(* CODESYS project sensata_utilities.library
   Company: Sensata Technologies
   Version: 0.0.1
   DocFormat: reStructuredText
   Placeholder: Sensata_Utilities
   Title: Sensata_Utilities

Project tree, tasks and I/O mapping:
  libraries: Sensata_Common, * (Sensata Technologies); Tc2_Standard, * (Beckhoff Automation GmbH); Tc2_System, * (Beckhoff Automation GmbH); Tc2_Utilities, * (Beckhoff Automation GmbH); Tc3_JsonXml, * (Beckhoff Automation GmbH); Tc3_Module, * (Beckhoff Automation GmbH)
  Abstract/
    Obsolete/
      function block FB_DeviceAPI [ST]: M_Connect, M_Disconnect, M_GetConnectStatus, P_bConnectBusy, P_bConnected, M_CallMethod, M_GetProperty, P_bDeviceInterfaceBusy
    function block FB_CommandRouter [ST]: M_Connect, M_Disconnect, M_GetConnectStatus, P_bConnectBusy, P_bConnected, M_AwaitCommand, M_RequestRoute, M_RouteCommand, P_bCommandRoutingBusy
  Concrete/
    Obsolete/
      function block FB_AdsDeviceAPI [ST]: M_CallMethod, M_GetProperty, P_bDeviceInterfaceBusy
    function block FB_AdsCommandRouter [ST]: M_BuildMessage, M_ParseResult, M_RouteCommand, P_bCommandRoutingBusy
    function block FB_ApiParamBuilder [ST]: M_AddArrayElement, M_AddParameter, M_AddStructMember, M_ClearParameters, M_OutputToParameterList, M_Add, M_Pushback, M_ParseBool, M_ParseDateTime, M_ParseDouble, M_ParseInt, M_ParseInt64, M_ParseString, M_ParseUint, M_ParseUint64, M_GetArrayElement, M_GetParameter, M_GetStructMember, M_LoadFromParameterList
  DUTs/
    Obsolete/
      data type T_ApiMethodParameters
    data type E_AdsCommandRouterError
    data type ST_ApiParameter
    data type T_ApiMessage
    data type T_ApiParameterList
    data type T_ApiParamValue
  Globals/
    Obsolete/
      global variables GVL_DeviceAPI
    global variables GVL_Api
  Interfaces/
    Obsolete/
      interface I_DeviceInterface: M_CallMethod, M_GetProperty, P_bDeviceInterfaceBusy
      interface I_ModularAPI: M_CallMethod, P_bApiBusy
    interface I_CommandRouting: M_AwaitCommand, M_RequestRoute, M_RouteCommand, P_bCommandRoutingBusy
  Project Information/
    function F_GetCompany [ST]
    function F_GetTitle [ST]
    function F_GetVersion [ST]
  Version/
    global variables Global_Version
*)

// DUTs/Obsolete/T_ApiMethodParameters
{attribute 'obsolete' := 'Only used on obsolete FB_DeviceAPI'} 
TYPE T_ApiMethodParameters : 
	ARRAY [1..GVL_DeviceAPI.uintMAX_CALL_METHOD_PARAMETERS]
		OF ARRAY [1..2] OF Tc2_System.T_MaxString;
END_TYPE

// DUTs/E_AdsCommandRouterError
{attribute 'qualified_only'}
{attribute 'strict'}
TYPE E_AdsCommandRouterError :
(
	None := 0,
	IncorrectResponseFormat := 100,
	NoResponseReceived := 101,
	AdsError := 200,
	PointerError := 300
) UDINT;
END_TYPE

// DUTs/ST_ApiParameter
TYPE ST_ApiParameter :
STRUCT
	strKey : T_MaxString;
	strValue : T_ApiParamValue;
END_STRUCT
END_TYPE

// DUTs/T_ApiMessage
TYPE T_ApiMessage : STRING(GVL_Api.dintMSG_STRING_SIZE); END_TYPE

// DUTs/T_ApiParameterList
TYPE T_ApiParameterList : ARRAY[GVL_Api.dintPARAM_LOWER_BOUND..GVL_Api.dintPARAM_UPPER_BOUND] OF ST_ApiParameter; END_TYPE

// DUTs/T_ApiParamValue
TYPE T_ApiParamValue : STRING(GVL_Api.dintPARAM_STRING_SIZE); END_TYPE

// Globals/Obsolete/GVL_DeviceAPI
{attribute 'qualified_only'}
VAR_GLOBAL CONSTANT
	uintMAX_CALL_METHOD_PARAMETERS : UINT := 16;
END_VAR

// Globals/GVL_Api
{attribute 'qualified_only'}
VAR_GLOBAL CONSTANT
	dintPARAM_LOWER_BOUND : DINT := 0;
	dintPARAM_UPPER_BOUND : DINT := 31;
	dintPARAM_STRING_SIZE : DINT := 1023;
	dintMSG_STRING_SIZE : DINT := 4095;
END_VAR

// Version/Global_Version
{attribute 'TcGenerated'}
{attribute 'no-analysis'}
{attribute 'linkalways'}
// This function has been automatically generated from the project information.
VAR_GLOBAL CONSTANT
	{attribute 'const_non_replaced'}
	stLibVersion_Sensata_Utilities : ST_LibVersion := (iMajor := 0, iMinor := 0, iBuild := 1, iRevision := 0, nFlags := 0, sVersion := '0.0.1');
END_VAR

// Abstract/Obsolete/FB_DeviceAPI
(*
===============================================================================
Abstract Device API
===============================================================================
:Contact: Kevin Sanita <ksanita@sensata.com>
:Last Edited: March 2022

:Description: Represents a device API that allows for methods and
	properties to be called and accessed

:Notes:
* ``M_CallMethod`` to send a call method command to a device API
* ``M_GetProperty`` to send a get property command to a device API

:Change Log:
- **March 25, 2022** Initial version
*)
{attribute 'obsolete' := 'Use FB_CommandRouter instead!'} 
FUNCTION_BLOCK ABSTRACT FB_DeviceAPI EXTENDS FB_Module IMPLEMENTS I_DeviceInterface, I_Connectable
VAR_INPUT
END_VAR
VAR_OUTPUT
END_VAR
VAR
	bConnected: BOOL;
END_VAR

(* Connect to the device. *)
METHOD M_Connect : BOOL
bConnected := TRUE;
M_Connect := TRUE;
THIS^.M_LogWarning('M_Connect not implemented!');
END_METHOD

(* Disconnect from the camera. *)
METHOD M_Disconnect : BOOL
bConnected := FALSE;
M_Disconnect := TRUE;
THIS^.M_LogWarning('M_Disconnect not implemented!');
END_METHOD

(* Get the device connection status. *)
METHOD M_GetConnectStatus : BOOL
VAR_OUTPUT
	(* TRUE if the device is connected, FALSE otherwise. *)
	bConnected	: BOOL;
END_VAR
bConnected := THIS^.bConnected;
M_GetConnectStatus := TRUE;
END_METHOD

(* TRUE while the device is connecting or disconnecting. *)
PROPERTY P_bConnectBusy : BOOL
GET
P_bConnectBusy := FALSE;
END_GET
END_PROPERTY

(* TRUE if the camera is connected. *)
PROPERTY P_bConnected : BOOL
GET
P_bConnected := bConnected;
END_GET
END_PROPERTY

(* Calls a device method from a device API. *)
METHOD M_CallMethod : BOOL
VAR_INPUT
	(* UniqueID of the target module. *)
	strTargetId		: Tc2_System.T_MaxString;
	(* Name of the method to call. *)
	strMethodName	: Tc2_System.T_MaxString;
	(* 2D array of parameter name and parameter value. *)
	arrParameters	: T_ApiMethodParameters;
END_VAR
VAR_OUTPUT
	(* Return data of the method. *)
	strReturn	: Tc2_System.T_MaxString;
END_VAR
M_CallMethod := FALSE;
END_METHOD

(* Gets the value of a device property through an API. *)
METHOD M_GetProperty : BOOL
VAR_INPUT
	(* Name of the property to get. *)
	strPropertyName	: Tc2_System.T_MaxString;
END_VAR
VAR_OUTPUT
	(* Value of the property. *)
	strReturn	: Tc2_System.T_MaxString;
END_VAR
M_GetProperty := FALSE;
END_METHOD

(* True while a device interface command is running. *)
PROPERTY P_bDeviceInterfaceBusy : BOOL
GET
P_bDeviceInterfaceBusy := FALSE;
END_GET
END_PROPERTY

END_FUNCTION_BLOCK

// Abstract/FB_CommandRouter
FUNCTION_BLOCK FB_CommandRouter EXTENDS FB_Module
	IMPLEMENTS I_CommandRouting, I_Connectable
VAR_INPUT
END_VAR
VAR_OUTPUT
END_VAR
VAR
	cr_bConnected: BOOL;
END_VAR

(* This method should establish any external connections required to use the
	functions of the device, and return TRUE and set P_bConnected to TRUE once
	connected. *)
METHOD M_Connect : BOOL
THIS^.M_LogWarning('M_Connect not implemented!');
cr_bConnected := TRUE;
M_Connect := TRUE;
END_METHOD

(* This method should break any connections established by M_Connect. It should
	immediately set P_bConnected to false unless all connections are known to
	be still active, and return TRUE once those connections are all fully
	disconnected. *)
METHOD M_Disconnect : BOOL
THIS^.M_LogWarning('M_Disconnect not implemented!');
cr_bConnected := FALSE;
M_Disconnect := TRUE;
END_METHOD

(* This method should explicitly check the connection status of the device.
	Once the connection status is known, this method should return TRUE.
	If this method fails, P_bConnected should be set to FALSE since the device
	is not absolutely known to still be connected. *)
METHOD M_GetConnectStatus : BOOL
VAR_OUTPUT
	(* This should return TRUE if all connections required to make the device
		function properly are known to be connected, and FALSE otherwise. *)
	bConnected	: BOOL;
END_VAR
THIS^.M_LogWarning('M_GetConnectStatus not implemented!');
M_GetConnectStatus := TRUE;
bConnected := cr_bConnected;
END_METHOD

(* This property should be TRUE while any method in this interface is actively
	executing, or FALSE otherwise. *)
PROPERTY P_bConnectBusy : BOOL
GET
P_bConnectBusy := FALSE;
END_GET
END_PROPERTY

(* This should be set to TRUE if M_Connect is successful or M_GetConnectStatus
	determines the device to be connected, and set to FALSE if M_Disconnect is
	called at all, M_GetConnectStatus fails, or M_GetConnectStatus determines
	the device to be not connected. *)
PROPERTY P_bConnected : BOOL
GET
P_bConnected := cr_bConnected;
END_GET
END_PROPERTY

(* Waits for the command with the given route ID to complete. *)
METHOD M_AwaitCommand : BOOL
VAR_INPUT
	(* ID assigned to the route. *)
	_in_udintRouteId	: UDINT;
	(* Timeout time for the command. *)
	_in_timeTimeout	: TIME;
END_VAR
VAR_IN_OUT
	(* Array of data key:value pairs. This will be filled with output
		data on command success. This is required due to memory limitations
		within Beckhoff. *)
	_inout_arrOutputs	: T_ApiParameterList;
END_VAR
VAR_OUTPUT
	(* True if the command executed without error. Does not necessarily
	mean the command performed the task it was expected to perform, just
	means that the method returned a value. *)
	_out_bCommandExecuted	: BOOL;
	(* The return value of the method. *)
	_out_strReturnValue	: T_ApiParamValue;
END_VAR
THIS^.M_LogWarning('M_AwaitCommand not implemented!');
M_AwaitCommand := TRUE;
END_METHOD

(* Sends a route request and returns a route ID if successfully routed. 
Use M_AwaitCommand with the route ID as input in order to wait for and get
the results of the routed command. *)
METHOD M_RequestRoute : BOOL
VAR_INPUT
	(* Unique ID of the module to call the command on. *)
	_in_strModuleId	: Tc2_System.T_MaxString;
	(* Name of the method to call. *)
	_in_strMethodName	: Tc2_System.T_MaxString;
	(* Timeout time for the route. *)
	_in_timeTimeout	: TIME;
END_VAR
VAR_IN_OUT
	(* Array of data key:value pairs. This should be set to the parameters
		of the command. *)
	_inout_arrParameters	: T_ApiParameterList;
END_VAR
VAR_OUTPUT
	(* ID assigned to the route. *)
	_out_udintRouteId	: UDINT;
END_VAR
THIS^.M_LogWarning('M_RequestRoute not implemented!');
M_RequestRoute := TRUE;
END_METHOD

(* Routes the given command and waits for the command to finish before
returning the output data of the command. *)
METHOD M_RouteCommand : BOOL
VAR_INPUT
	(* Unique ID of the module to call the command on. *)
	_in_strModuleId	: Tc2_System.T_MaxString;
	(* Name of the method to call. *)
	_in_strMethodName	: Tc2_System.T_MaxString;
	(* Timeout time for the command. *)
	_in_timeTimeout	: TIME;
END_VAR
VAR_IN_OUT
	(* Array of input parameter key:value pairs. *)
	_inout_arrParameters	: T_ApiParameterList;
	(* Array of output key:value pairs. Will be cleared and then populated with output data. *)
	_inout_arrOutputs	: T_ApiParameterList;
END_VAR
VAR_OUTPUT
	(* True if the command executed without error. Does not necessarily
	mean the command performed the task it was expected to perform, just
	means that the method returned a value. *)
	_out_bCommandExecuted	: BOOL;
	(* The return value of the method as a string. *)
	_out_strReturnValue	: T_ApiParamValue;
END_VAR
THIS^.M_LogWarning('M_RouteCommand not implemented!');
M_RouteCommand := TRUE;
END_METHOD

(* TRUE while any method in this interface is running. *)
PROPERTY P_bCommandRoutingBusy : BOOL
GET
P_bCommandRoutingBusy := TRUE;
END_GET
END_PROPERTY

END_FUNCTION_BLOCK

// Interfaces/I_CommandRouting
INTERFACE I_CommandRouting

(* Waits for the command with the given route ID to complete. *)
METHOD M_AwaitCommand : BOOL
VAR_INPUT
	(* ID assigned to the route. *)
	_in_udintRouteId : UDINT;
	
	(* Timeout time for the command. *)
	_in_timeTimeout : TIME;
END_VAR
VAR_IN_OUT
	(* Array of data key:value pairs. This will be filled with output
		data on command success. This is required due to memory limitations
		within Beckhoff. *)
	_inout_arrOutputs : T_ApiParameterList;
END_VAR
VAR_OUTPUT
	(* True if the command executed without error. Does not necessarily
	mean the command performed the task it was expected to perform, just
	means that the method returned a value. *)
	_out_bCommandExecuted : BOOL;
	
	(* The return value of the method. *)
	_out_strReturnValue : T_ApiParamValue;
END_VAR
END_METHOD

(* Sends a route request and returns a route ID if successfully routed. 
Use M_AwaitCommand with the route ID as input in order to wait for and get
the results of the routed command. *)
METHOD M_RequestRoute : BOOL
VAR_INPUT
	(* Unique ID of the module to call the command on. *)
	_in_strModuleId : T_MaxString;
	
	(* Name of the method to call. *)
	_in_strMethodName : T_MaxString;
	
	(* Timeout time for the route. *)
	_in_timeTimeout : TIME;
END_VAR
VAR_IN_OUT
	(* Array of data key:value pairs. This should be set to the parameters
		of the command. *)
	_inout_arrParameters : T_ApiParameterList;
END_VAR
VAR_OUTPUT
	(* ID assigned to the route. *)
	_out_udintRouteId : UDINT;
END_VAR
END_METHOD

(* Routes the given command and waits for the command to finish before
returning the output data of the command. *)
METHOD M_RouteCommand : BOOL
VAR_INPUT
	(* Unique ID of the module to call the command on. *)
	_in_strModuleId	: Tc2_System.T_MaxString;
	
	(* Name of the method to call. *)
	_in_strMethodName	: Tc2_System.T_MaxString;
	
	(* Timeout time for the command. *)
	_in_timeTimeout	: TIME;
END_VAR
VAR_IN_OUT
	(* Array of input parameter key:value pairs. *)
	_inout_arrParameters	: T_ApiParameterList;
	
	(* Array of output key:value pairs. Will be cleared and then populated with output data. *)
	_inout_arrOutputs	: T_ApiParameterList;
END_VAR
VAR_OUTPUT
	(* True if the command executed without error. Does not necessarily
	mean the command performed the task it was expected to perform, just
	means that the method returned a value. *)
	_out_bCommandExecuted	: BOOL;
	
	(* The return value of the method as a string. *)
	_out_strReturnValue	: T_ApiParamValue;
END_VAR
END_METHOD

(* TRUE while any method in this interface is running. *)
PROPERTY P_bCommandRoutingBusy : BOOL
GET
END_GET
END_PROPERTY

END_INTERFACE

// Interfaces/Obsolete/I_DeviceInterface
INTERFACE I_DeviceInterface

(* Calls a device method from a device API. *)
METHOD M_CallMethod : BOOL
VAR_INPUT
	(* UniqueID of the target module. *)
	strTargetId		: Tc2_System.T_MaxString;
		
	(* Name of the method to call. *)
	strMethodName : T_MaxString;
	
	(* 2D array of parameter name and parameter value. *)
	arrParameters : T_ApiMethodParameters;
END_VAR
VAR_OUTPUT
	(* Return data of the method. *)
	strReturn : T_MaxString;
END_VAR
END_METHOD

(* Gets the value of a device property through an API. *)
METHOD M_GetProperty : BOOL
VAR_INPUT
	(* Name of the property to get. *)
	strPropertyName : T_MaxString;
END_VAR
VAR_OUTPUT
	(* Value of the property. *)
	strReturn : T_MaxString;
END_VAR
END_METHOD

(* True while a device interface command is running. *)
PROPERTY P_bDeviceInterfaceBusy : BOOL
GET
END_GET
END_PROPERTY

END_INTERFACE

// Concrete/Obsolete/FB_AdsDeviceAPI
(*
===============================================================================
ADS Device API
===============================================================================
:Contact: Kevin Sanita <ksanita@sensata.com>
:Last Edited: March 2022

:Description: Represents a device API that allows for methods and
	properties to be called and accessed through ADS

:Notes:
* ``M_CallMethod`` to send a call method command to a device API through ADS
* ``M_GetProperty`` to send a get property command to a device API through ADS

:Change Log:
- **March 25, 2022** Initial version
*)
{attribute 'obsolete' := 'Use FB_AdsCommandRouter instead!'} 
FUNCTION_BLOCK FB_AdsDeviceAPI EXTENDS FB_DeviceAPI IMPLEMENTS I_DeviceInterface
VAR_INPUT
	(* ADS address of the device ADS server. *)
	strAdsAddress: T_AmsNetId;
	
	(* ADS port of the device ADS server. *)
	udintAdsPort: T_AmsPort;
	
	(* Optional timeout for the ADS commands. Default 60 seconds. *)
	timeAdsTimeout: TIME := T#60S;
END_VAR
VAR_OUTPUT
END_VAR
VAR CONSTANT
	udintGET_PROPERTY_GROUP : UDINT := 16#1000;
	udintGET_PROPERTY_OFFSET : UDINT := 0;
	udintCALL_METHOD_GROUP : UDINT := 16#2000;
	udintCALL_METHOD_OFFSET : UDINT := 0;
END_VAR
VAR
	fbAds: ADSRDWRTEX;
	udintGroup: UDINT;
	udintOffset: UDINT;
	strMessage: T_MaxString;
	bSend: BOOL;
	udintAdsReadByteCount: UDINT;
	strResponse: T_MaxString;
	bAdsBusy: BOOL;
	udintAdsErrorId: UDINT;
	bBusy: BOOL;
	bAdsError: BOOL;
	fbJson: FB_JsonDomParser;
	intCallMethodStep: INT;
	intGetPropertyStep: INT;
END_VAR

fbAds(
	NETID:= strAdsAddress, 
	PORT:= udintAdsPort, 
	IDXGRP:= udintGroup, 
	IDXOFFS:= udintOffset, 
	WRITELEN:= INT_TO_UDINT(LEN(strMessage)), 
	READLEN:= SIZEOF(T_MaxString), 
	SRCADDR:= ADR(strMessage), 
	DESTADDR:= ADR(strResponse), 
	WRTRD:= bSend, 
	TMOUT:= timeAdsTimeout, 
	BUSY=> bAdsBusy, 
	ERR=> bAdsError, 
	ERRID=> udintAdsErrorId, 
	COUNT_R=> udintAdsReadByteCount);
	
bSend := FALSE;

(* Calls a device method from a device API. *)
METHOD M_CallMethod : BOOL
VAR_INPUT
	(* UniqueID of the target module. *)
	strTargetId		: Tc2_System.T_MaxString;
	(* Name of the method to call. *)
	strMethodName	: Tc2_System.T_MaxString;
	(* 2D array of parameter name and parameter value. *)
	arrParameters	: T_ApiMethodParameters;
END_VAR
VAR_OUTPUT
	(* Return data of the method. *)
	strReturn	: Tc2_System.T_MaxString;
END_VAR

VAR
	strCommand : T_MaxString;
	jsonParams: Tc3_JsonXml.PVOID;
	dintParamIndex: DINT;
	jsonMsg: Tc3_JsonXml.PVOID;
END_VAR
M_CallMethod := FALSE;
CASE intCallMethodStep OF
	0:
		IF NOT bAdsBusy AND NOT bBusy AND NOT P_bError THEN
			bBusy := TRUE;
			THIS^.M_LogMessage('Calling ADS method');
			
			// Generate JSON message
			jsonMsg := fbJson.ParseDocument('{}');
			fbJson.AddStringMember(jsonMsg, 'Target', strTargetId);			
			fbJson.AddStringMember(jsonMsg, 'Name', strMethodName);
			jsonParams := fbJson.AddObjectMember(jsonMsg, 'Params');
			FOR dintParamIndex := 1 TO GVL_DeviceAPI.uintMAX_CALL_METHOD_PARAMETERS DO
				IF LEN(arrParameters[dintParamIndex][1]) > 0 THEN
					fbJson.AddStringMember(
						jsonParams,
						arrParameters[dintParamIndex][1],
						arrParameters[dintParamIndex][2]);
				END_IF
			END_FOR
			strCommand := fbJson.GetDocument();
			
			// Set command parameters
			bSend := FALSE;
			strMessage := strCommand;
			udintGroup := udintCALL_METHOD_GROUP;
			udintOffset := udintCALL_METHOD_OFFSET;
			
			MEMSET(ADR(strResponse),0,SIZEOF(strResponse));
			// Go to next step
			intCallMethodStep := 10;
		END_IF
		
	10:
		// Wait for ADS to start running
		bSend := TRUE;
		IF bAdsBusy THEN
			intCallMethodStep := 20;
		END_IF
		
	20:
		IF NOT bAdsBusy THEN
			udintGroup := 0;
			udintOffset := 0;
			bSend := FALSE;
			IF bAdsError THEN
				THIS^.M_SetError(
					udintAdsErrorId,
					'ADS error while trying to call method!');
			ELSE
				THIS^.M_LogMessage(CONCAT('Received method response: ', strResponse));
				strReturn := strResponse;
				M_CallMethod := TRUE;
			END_IF
			bBusy := FALSE;
			intCallMethodStep := 0;
		END_IF
END_CASE
END_METHOD

(* Gets the value of a device property through an API. *)
METHOD M_GetProperty : BOOL
VAR_INPUT
	(* Name of the property to get. *)
	strPropertyName	: Tc2_System.T_MaxString;
END_VAR
VAR_OUTPUT
	(* Value of the property. *)
	strReturn	: Tc2_System.T_MaxString;
END_VAR
M_GetProperty := FALSE;
CASE intGetPropertyStep OF
	0:
		IF NOT bAdsBusy AND NOT bBusy AND NOT P_bError THEN
			bBusy := TRUE;
			THIS^.M_LogMessage('Getting property over ADS');
			
			// Set command parameters
			bSend := FALSE;
			strMessage := strPropertyName;
			udintGroup := udintGET_PROPERTY_GROUP;
			udintOffset := udintGET_PROPERTY_OFFSET;
			
			// Go to next step
			intGetPropertyStep := 10;
		END_IF
		
	10:
		// Wait for ADS to start running
		bSend := TRUE;
		IF bAdsBusy THEN
			intGetPropertyStep := 20;
		END_IF
		
	20:
		IF NOT bAdsBusy THEN
			udintGroup := 0;
			udintOffset := 0;
			bSend := FALSE;
			IF bAdsError THEN
				THIS^.M_SetError(
					udintAdsErrorId,
					'ADS error while trying to get property!');
			ELSE
				THIS^.M_LogMessage(CONCAT('Received property response: ', strResponse));
				strReturn := strResponse;
				M_GetProperty := TRUE;
			END_IF
			bBusy := FALSE;
			intGetPropertyStep := 0;
		END_IF
END_CASE
END_METHOD

(* True while a device interface command is running. *)
PROPERTY P_bDeviceInterfaceBusy : BOOL
GET
P_bDeviceInterfaceBusy := bBusy;
END_GET
END_PROPERTY

END_FUNCTION_BLOCK

// Concrete/FB_AdsCommandRouter
(*
Concrete implementation of a command router that works over ADS.
*)
FUNCTION_BLOCK FB_AdsCommandRouter EXTENDS FB_CommandRouter
	IMPLEMENTS I_CommandRouting
VAR_INPUT
	(* AMS Net ID of the PC that the API is running on. *)
	in_strNetId: T_AmsNetId;
	(* Port address that the API's ADS Server is running on. *)
	in_uintPort: T_AmsPort;
END_VAR
VAR_OUTPUT
END_VAR
VAR
	bRouterBusy: BOOL; // True while the router is being used by a method
	bRouteCommandReset: BOOL;
	bRouteCommandBusy: BOOL;
END_VAR
VAR CONSTANT
	udintROUTE_GROUP: UDINT := 16#1000; // Index group of the route command
	udintAWAIT_GROUP: UDINT := 16#2000; // Index group of the get result command
	udintROUTE_AND_AWAIT_GROUP: UDINT := 16#4000; // Index group of the route and return command
END_VAR

// Reset router step if route command stops being called prematurely
IF NOT bRouteCommandBusy THEN
	bRouteCommandReset := TRUE;
	//THIS^.M_LogWarning('M_RouteCommand stopped being called prematurely!');
END_IF
bRouteCommandBusy := FALSE;

(* Builds the message string from input variables. *)
METHOD PRIVATE M_BuildMessage : BOOL
VAR_INPUT
	(* Unique ID of the module to call the command on. *)
	_in_strModuleId	: Tc2_System.T_MaxString;
	(* Name of the method to call. *)
	_in_strMethodName	: Tc2_System.T_MaxString;
END_VAR
VAR_IN_OUT
	(* Array of parameter key:value pairs. *)
	_inout_arrParameters : T_ApiParameterList;
END_VAR
VAR_OUTPUT
	(* Message string. *)
	_out_strMessage: T_ApiMessage;
END_VAR
VAR_INST
	_inst_fbJson: FB_JsonDynDomParser; // JSON parser function block
END_VAR
VAR
	_pJsonDoc: Tc3_JsonXml.PVOID; // Pointer to the JSON document
	_pJsonModuleId: Tc3_JsonXml.PVOID; // Pointer to the JSON module ID member
	_pJsonMethodName: Tc3_JsonXml.PVOID; // Pointer to the JSON method name member
	_pJsonParameters: Tc3_JsonXml.PVOID; // Pointer to the JSON parameters member
	_dintParamIndex: DINT; // Current parameter index
	_stParameter: ST_ApiParameter; // Current parameter being added to the JSON doc
END_VAR
// Create a blank JSON object
_pJsonDoc := _inst_fbJson.NewDocument();

// Add module ID and method name
_pJsonModuleId := _inst_fbJson.AddStringMember(_pJsonDoc, 'ModuleId', _in_strModuleId);
_pJsonMethodName := _inst_fbJson.AddStringMember(_pJsonDoc, 'MethodName', _in_strMethodName);

// Add each parameter with a key in the parameters array
_pJsonParameters := _inst_fbJson.AddObjectMember(_pJsonDoc, 'Parameters');
FOR _dintParamIndex := GVL_Api.dintPARAM_LOWER_BOUND TO GVL_Api.dintPARAM_UPPER_BOUND DO
	_stParameter := _inout_arrParameters[_dintParamIndex];
	IF LEN(_stParameter.strKey) > 0 THEN
		_inst_fbJson.AddJsonMember(_pJsonParameters, _stParameter.strKey, _stParameter.strValue);
	END_IF
END_FOR

// Output the document to strMessage
MEMSET(ADR(_out_strMessage),0,SIZEOF(_out_strMessage));
_inst_fbJson.CopyDocument(_out_strMessage, SIZEOF(_out_strMessage));

// Return true
M_BuildMessage := TRUE;
END_METHOD

METHOD PRIVATE M_ParseResult : BOOL
VAR_INPUT
	(* Result message from the API. *)
	_in_strResult: T_ApiMessage;
END_VAR
VAR_IN_OUT
	(* Any output values of the command. *)
	_inout_arrOutputs	: T_ApiParameterList;
END_VAR
VAR_OUTPUT
	(* True if the command executed without error. *)
	_out_bCommandExecuted	: BOOL;
	(* The return value of the method. *)
	_out_strReturnValue	: T_ApiParamValue;
END_VAR
VAR_INST
	_inst_fbJson: FB_JsonDynDomParser; // JSON parser function block
END_VAR
VAR
	_pJsonDoc: Tc3_JsonXml.PVOID; // Pointer to the JSON document
	_pJsonSucceeded: Tc3_JsonXml.PVOID; // Pointer to the "Successful" member
	_pJsonReturnValue: Tc3_JsonXml.PVOID; // Pointer to the "ReturnData" member
	_pJsonOutput: Tc3_JsonXml.PVOID; // Pointer to the "OutputData" member
	_pJsonIterator: Tc3_JsonXml.PVOID; // Iterator for the output data
	_pJsonIteratorEnd: Tc3_JsonXml.PVOID; // End pointer for the output data iterator
	_dintParamIndex: DINT; // Output data index
	_pOutputValue: Tc3_JsonXml.PVOID; // Pointer to the current output data value
	_strValue: T_ApiParamValue; // Output data value as a JSON string
END_VAR
// Parse the JSON string as a JSON document
_pJsonDoc := _inst_fbJson.ParseDocument(_in_strResult);

// Get success status
_pJsonSucceeded := _inst_fbJson.FindMember(_pJsonDoc, 'Successful');

// Parse the success status
IF (_pJsonSucceeded > 0) THEN
	_out_bCommandExecuted := _inst_fbJson.GetBool(_pJsonSucceeded);
	
// Throw an error if no success status member in the JSON
ELSE
	IF NOT THIS^.P_bError THEN
		THIS^.M_SetError(
			E_AdsCommandRouterError.IncorrectResponseFormat,
			'Incorrect response format from the API!');
	END_IF
END_IF

// Get return value
_pJsonReturnValue := _inst_fbJson.FindMember(_pJsonDoc, 'ReturnData');

// If there is return data, parse it
IF (_pJsonReturnValue > 0) THEN
	_inst_fbJson.CopyJson(_pJsonReturnValue, _out_strReturnValue, SIZEOF(_out_strReturnValue));
	
// Throw an error if the command executed but there is no return data
ELSIF _out_bCommandExecuted THEN
	IF NOT THIS^.P_bError THEN
		THIS^.M_SetError(
			E_AdsCommandRouterError.IncorrectResponseFormat,
			'Incorrect response format from the API!');
	END_IF
END_IF

// Get output data
_pJsonOutput := _inst_fbJson.FindMember(_pJsonDoc, 'OutputData');

// If there is output data, parse it
IF (_pJsonOutput > 0) THEN
	
	// Clear output array
	FOR _dintParamIndex := GVL_Api.dintPARAM_LOWER_BOUND TO GVL_Api.dintPARAM_UPPER_BOUND DO
		_inout_arrOutputs[_dintParamIndex].strKey := '';
		MEMSET(ADR(_inout_arrOutputs[_dintParamIndex].strValue),0,SIZEOF(_inout_arrOutputs[_dintParamIndex].strValue));
	END_FOR
	
	// Initialize output data iterator and index
	_pJsonIterator := _inst_fbJson.MemberBegin(_pJsonOutput);
	_pJsonIteratorEnd := _inst_fbJson.MemberEnd(_pJsonOutput);
	_dintParamIndex := GVL_Api.dintPARAM_LOWER_BOUND;
	
	// Populate output data array with data from the JSON response data
	WHILE _pJsonIterator <> _pJsonIteratorEnd AND _dintParamIndex <= GVL_Api.dintPARAM_UPPER_BOUND DO
		// Populate the output array with the name of the current member
		_inout_arrOutputs[_dintParamIndex].strKey := _inst_fbJson.GetMemberName(_pJsonIterator);
		
		// Get the pointer to the value of the current member
		_pOutputValue := _inst_fbJson.GetMemberValue(_pJsonIterator);
		
		// Get the value as a JSON string
		_inst_fbJson.CopyJson(_pOutputValue, _strValue, SIZEOF(_strValue));
		
		// Populate the output array with the JSON string of the value
		_inout_arrOutputs[_dintParamIndex].strValue := _strValue;
		
		// Increment iterator and index
		_pJsonIterator := _inst_fbJson.NextMember(_pJsonIterator);
		_dintParamIndex := _dintParamIndex + 1;
	END_WHILE

// Throw an error if command executed but no output data member in the response JSON	
ELSIF _out_bCommandExecuted THEN
	IF NOT THIS^.P_bError THEN
		THIS^.M_SetError(
			E_AdsCommandRouterError.IncorrectResponseFormat,
			'Incorrect response format from the API!');
	END_IF
END_IF

// Return true
M_ParseResult := TRUE;
END_METHOD

(* Routes the given command and waits for the command to finish before
returning the output data of the command. *)
METHOD M_RouteCommand : BOOL
VAR_INPUT
	(* Unique ID of the module to call the command on. *)
	_in_strModuleId	: Tc2_System.T_MaxString;
	(* Name of the method to call. *)
	_in_strMethodName : Tc2_System.T_MaxString;
	(* Timeout time for the command. *)
	_in_timeTimeout	: TIME;
END_VAR
VAR_IN_OUT
	(* Array of input parameter key:value pairs. *)
	_inout_arrParameters	: T_ApiParameterList;
	(* Array of output key:value pairs. Will be cleared and then populated with output data. *)
	_inout_arrOutputs	: T_ApiParameterList;
END_VAR
VAR_OUTPUT
	(* True if the command executed without error. Does not necessarily
	mean the command performed the task it was expected to perform, just
	means that the method returned a value. *)
	_out_bCommandExecuted	: BOOL;
	(* The return value of the method as a string. *)
	_out_strReturnValue	: T_ApiParamValue;
END_VAR
VAR_INST
	_inst_strMessage: T_ApiMessage; // JSON message that gets sent to the API
	_inst_strOutput: T_ApiMessage; // JSON message with route results received from the API
	_inst_pAds: POINTER TO ADSRDWRTEX; // Beckhoff's ADS read/write command function block
	_inst_bBusy: BOOL; // TRUE if the ADS function block is busy
	_inst_bErr: BOOL; // TRUE if the ADS function block has an error
	_inst_udintErrId: UDINT; // Error ID from the ADS function block if it has an error
	_inst_bWait: BOOL;
	_inst_uintStep: UINT;
END_VAR
VAR
	_udintReadCount: UDINT; // Size of the ADS read response in bytes
	_bMessageBuilt: BOOL; // Goes high once the build message method finishes
	_udintCleared: UDINT; // Number of bytes set when clearing the output string
	_bResultParsed: BOOL; // TRUE once the result parsing method finishes
	_bErrorSet: BOOL; // TRUE once an error is set on the FB
	_strBuiltMessage: T_ApiMessage; // Output of the build command method

END_VAR
VAR_INST // added by the converter: edge detectors and wires of the graphical bodies
    _w1, _w2, _w3, _w4, _w5, _w6, _w7, _w8, _w9, _w10, _w11, _w12, _w13, _w14, _w15, _w16, _w17, _w18, _w19 : BOOL;
END_VAR
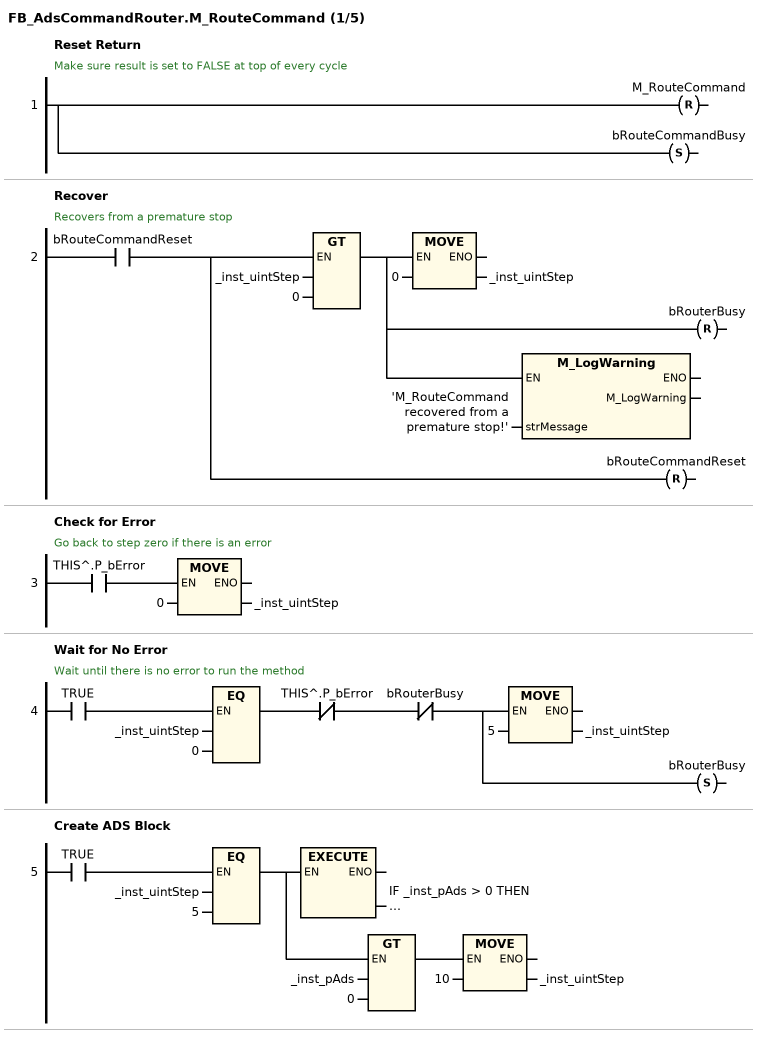
// NETWORK 1: Reset Return
// Make sure result is set to FALSE at top of every cycle
M_RouteCommand R= TRUE;
bRouteCommandBusy S= TRUE;

// NETWORK 2: Recover
// Recovers from a premature stop
_w1 := bRouteCommandReset;
_w2 := _w1 AND _inst_uintStep > 0;
IF _w2 THEN _inst_uintStep := 0; END_IF
bRouterBusy R= _w2;
IF _w2 THEN M_LogWarning(strMessage := 'M_RouteCommand recovered from a premature stop!'); END_IF
bRouteCommandReset R= _w1;

// NETWORK 3: Check for Error
// Go back to step zero if there is an error
IF THIS^.P_bError THEN _inst_uintStep := 0; END_IF

// NETWORK 4: Wait for No Error
// Wait until there is no error to run the method
_w3 := _inst_uintStep = 0 AND NOT THIS^.P_bError AND NOT bRouterBusy;
IF _w3 THEN _inst_uintStep := 5; END_IF
bRouterBusy S= _w3;

// NETWORK 5: Create ADS Block
_w4 := _inst_uintStep = 5;
IF _w4 THEN
    IF _inst_pAds > 0 THEN
    	__DELETE(_inst_pAds);
    	THIS^.M_LogWarning('Deleted old ADSRDWRTEX block. Could cause errors!');
    END_IF
    _inst_pAds := __NEW(ADSRDWRTEX);
END_IF
IF _w4 AND _inst_pAds > 0 THEN _inst_uintStep := 10; END_IF

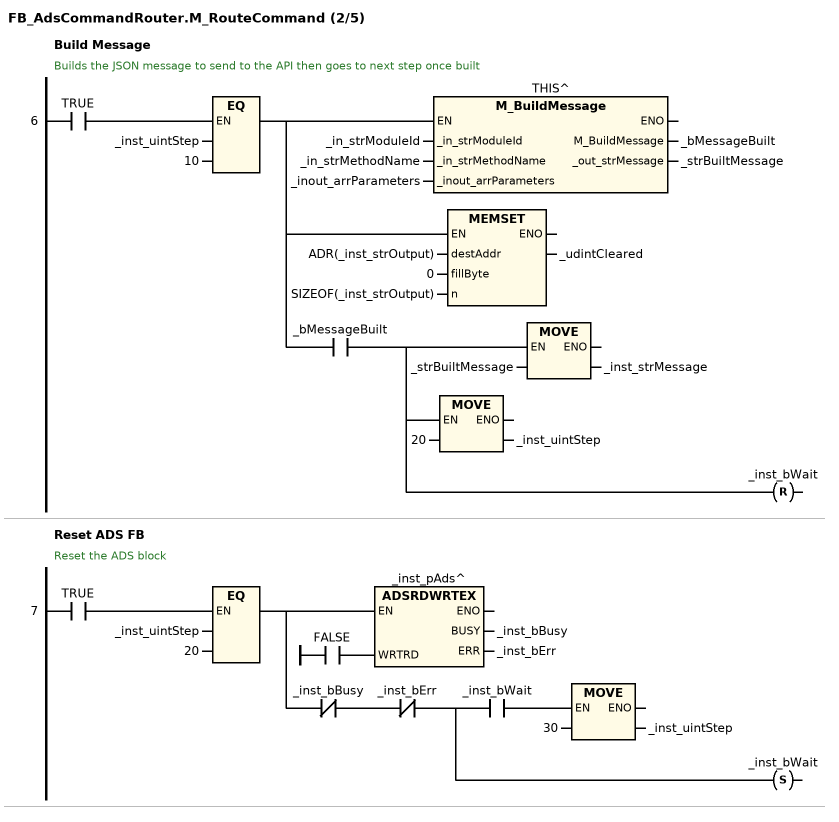
// NETWORK 6: Build Message
// Builds the JSON message to send to the API then goes to next step once built
_w5 := _inst_uintStep = 10;
IF _w5 THEN
    THIS^.M_BuildMessage(
        _in_strModuleId := _in_strModuleId,
        _in_strMethodName := _in_strMethodName,
        _inout_arrParameters := _inout_arrParameters,
        M_BuildMessage => _bMessageBuilt,
        _out_strMessage => _strBuiltMessage);
END_IF
IF _w5 THEN
    _udintCleared := MEMSET(destAddr := ADR(_inst_strOutput), fillByte := 0, n := SIZEOF(_inst_strOutput));
END_IF
_w6 := _w5 AND _bMessageBuilt;
IF _w6 THEN _inst_strMessage := _strBuiltMessage; END_IF
IF _w6 THEN _inst_uintStep := 20; END_IF
_inst_bWait R= _w6;

// NETWORK 7: Reset ADS FB
// Reset the ADS block
_w7 := _inst_uintStep = 20;
IF _w7 THEN
    _inst_pAds^(WRTRD := FALSE, BUSY => _inst_bBusy, ERR => _inst_bErr); // ADSRDWRTEX
END_IF
_w8 := _w7 AND NOT _inst_bBusy AND NOT _inst_bErr;
IF _w8 AND _inst_bWait THEN _inst_uintStep := 30; END_IF
_inst_bWait S= _w8;

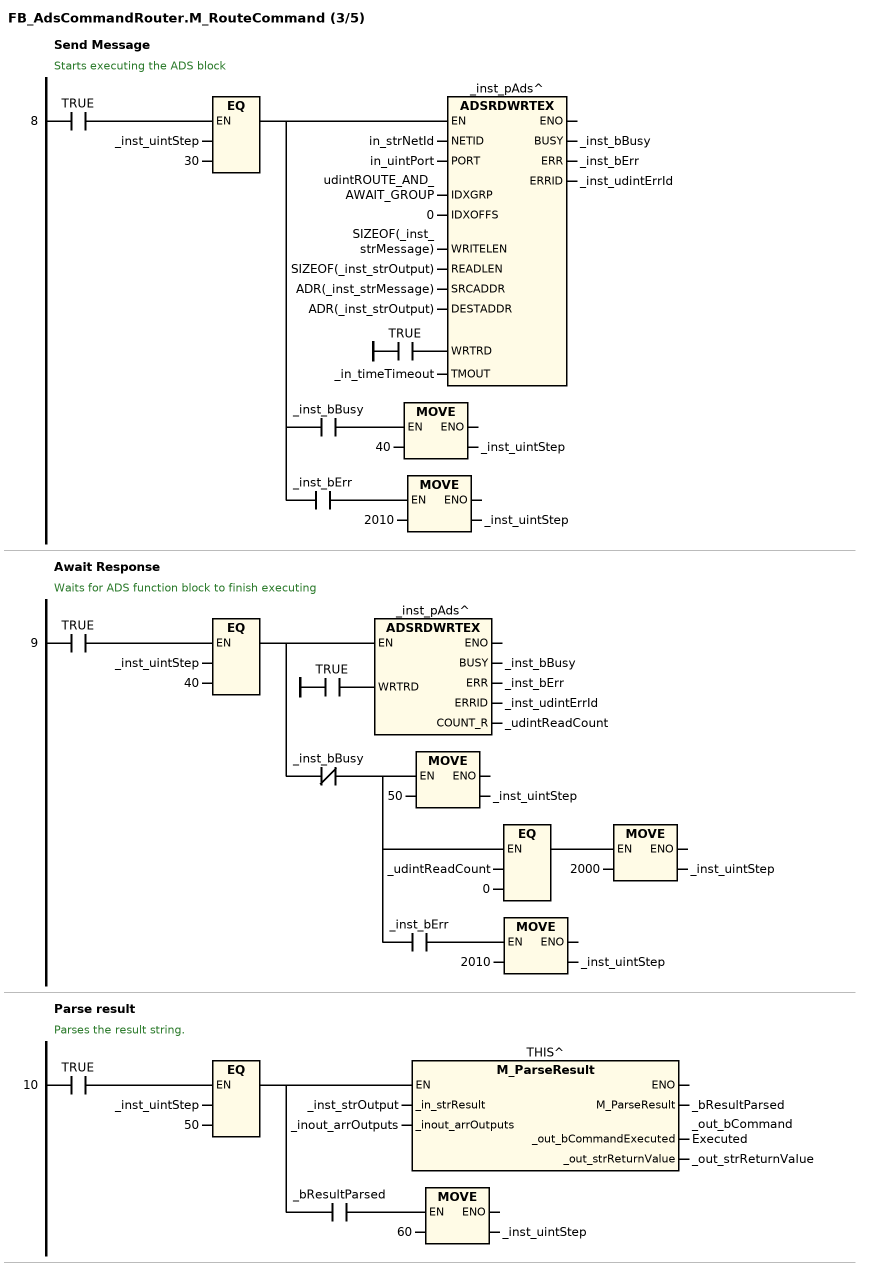
// NETWORK 8: Send Message
// Starts executing the ADS block
_w9 := _inst_uintStep = 30;
IF _w9 THEN
    _inst_pAds^(
        NETID := in_strNetId,
        PORT := in_uintPort,
        IDXGRP := udintROUTE_AND_AWAIT_GROUP,
        IDXOFFS := 0,
        WRITELEN := SIZEOF(_inst_strMessage),
        READLEN := SIZEOF(_inst_strOutput),
        SRCADDR := ADR(_inst_strMessage),
        DESTADDR := ADR(_inst_strOutput),
        WRTRD := TRUE,
        TMOUT := _in_timeTimeout,
        BUSY => _inst_bBusy,
        ERR => _inst_bErr,
        ERRID => _inst_udintErrId); // ADSRDWRTEX
END_IF
IF _w9 AND _inst_bBusy THEN _inst_uintStep := 40; END_IF
IF _w9 AND _inst_bErr THEN _inst_uintStep := 2010; END_IF

// NETWORK 9: Await Response
// Waits for ADS function block to finish executing
_w10 := _inst_uintStep = 40;
IF _w10 THEN
    _inst_pAds^(
        WRTRD := TRUE,
        BUSY => _inst_bBusy,
        ERR => _inst_bErr,
        ERRID => _inst_udintErrId,
        COUNT_R => _udintReadCount); // ADSRDWRTEX
END_IF
_w11 := _w10 AND NOT _inst_bBusy;
IF _w11 THEN _inst_uintStep := 50; END_IF
IF _w11 AND _udintReadCount = 0 THEN _inst_uintStep := 2000; END_IF
IF _w11 AND _inst_bErr THEN _inst_uintStep := 2010; END_IF

// NETWORK 10: Parse result
// Parses the result string.
_w12 := _inst_uintStep = 50;
IF _w12 THEN
    THIS^.M_ParseResult(
        _in_strResult := _inst_strOutput,
        _inout_arrOutputs := _inout_arrOutputs,
        M_ParseResult => _bResultParsed,
        _out_bCommandExecuted => _out_bCommandExecuted,
        _out_strReturnValue => _out_strReturnValue);
END_IF
IF _w12 AND _bResultParsed THEN _inst_uintStep := 60; END_IF

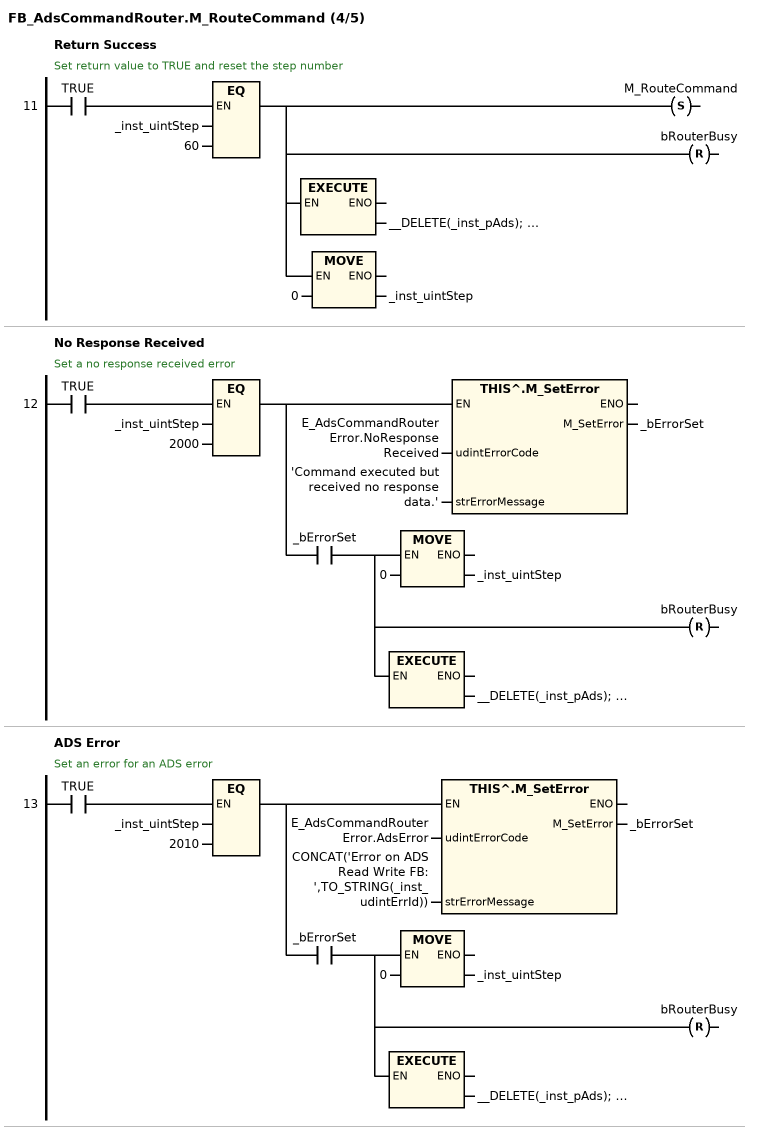
// NETWORK 11: Return Success
// Set return value to TRUE and reset the step number
_w13 := _inst_uintStep = 60;
M_RouteCommand S= _w13;
bRouterBusy R= _w13;
IF _w13 THEN __DELETE(_inst_pAds); END_IF
IF _w13 THEN _inst_uintStep := 0; END_IF

// NETWORK 12: No Response Received
// Set a no response received error
_w14 := _inst_uintStep = 2000;
IF _w14 THEN
    _bErrorSet := THIS^.M_SetError(udintErrorCode := E_AdsCommandRouterError.NoResponseReceived, strErrorMessage := 'Command executed but received no response data.');
END_IF
_w15 := _w14 AND _bErrorSet;
IF _w15 THEN _inst_uintStep := 0; END_IF
bRouterBusy R= _w15;
IF _w15 THEN __DELETE(_inst_pAds); END_IF

// NETWORK 13: ADS Error
// Set an error for an ADS error
_w16 := _inst_uintStep = 2010;
IF _w16 THEN
    _bErrorSet := THIS^.M_SetError(udintErrorCode := E_AdsCommandRouterError.AdsError, strErrorMessage := CONCAT('Error on ADS Read Write FB: ',TO_STRING(_inst_udintErrId)));
END_IF
_w17 := _w16 AND _bErrorSet;
IF _w17 THEN _inst_uintStep := 0; END_IF
bRouterBusy R= _w17;
IF _w17 THEN __DELETE(_inst_pAds); END_IF

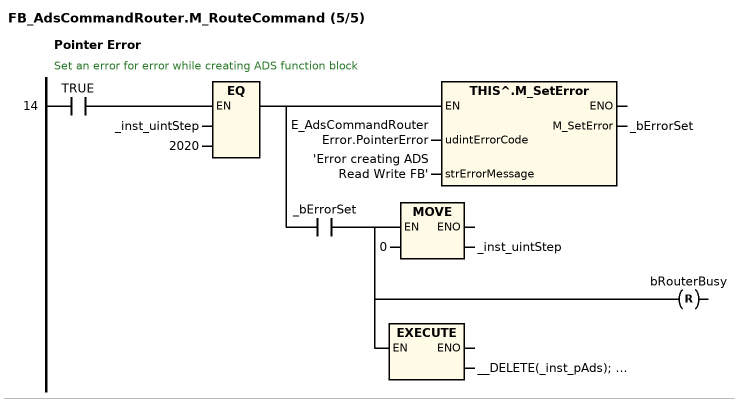
// NETWORK 14: Pointer Error
// Set an error for error while creating ADS function block
_w18 := _inst_uintStep = 2020;
IF _w18 THEN
    _bErrorSet := THIS^.M_SetError(udintErrorCode := E_AdsCommandRouterError.PointerError, strErrorMessage := 'Error creating ADS Read Write FB');
END_IF
_w19 := _w18 AND _bErrorSet;
IF _w19 THEN _inst_uintStep := 0; END_IF
bRouterBusy R= _w19;
IF _w19 THEN __DELETE(_inst_pAds); END_IF
END_METHOD

(* TRUE while any method in this interface is running. *)
PROPERTY P_bCommandRoutingBusy : BOOL
GET
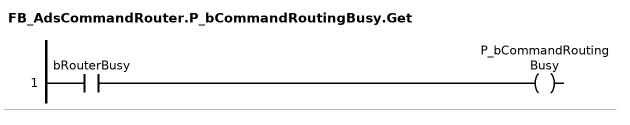
// NETWORK 1
P_bCommandRoutingBusy := bRouterBusy;
END_GET
END_PROPERTY

END_FUNCTION_BLOCK

// Concrete/FB_ApiParamBuilder
(*
Used to build an array of correctly-formatted ST_ApiParameter structs.

Use M_AddParameter to add a parameter to the parameters list.

If a parameter is a struct or array, use M_AddStructMember and M_AddArrayElement
respectively after M_AddParameter to manually build the struct or array in this
function block.

Use M_ClearParameters to clear the memory, and M_GetParameterList to get
the correctly formatted T_ApiParameters object.
*)
FUNCTION_BLOCK FB_ApiParamBuilder EXTENDS FB_Module
VAR_INPUT
END_VAR
VAR_OUTPUT
END_VAR
VAR
	fbJson : FB_JsonDynDomParser;
	pJsonDoc: Tc3_JsonXml.PVOID;
	bInitialized: BOOL := FALSE;
END_VAR

(* Appends a new element to the array given by the pointer and returns a
	pointer to the added value. Supports most primitive types directly.

	If the value is an array, will only add a blank array that must be populated
	manually by calling M_AddArrayElement with the pointer returned by this method. 

	If the value is a struct, will only add a blank struct that must be populated
	manually by calling M_AddStructMember with the pointer returned by this method. 

	Value will be stored as null if the value type is not yet supported. *)
METHOD M_AddArrayElement : PVOID
VAR_INPUT
	(* Pointer to the array that should be added to. This pointer is returned
		by any M_Add<item> methods that were used to add an array. *)
	_in_pArrayPointer : PVOID;
	
	(* The value to append to the array. *)
	_in_anyValue : ANY;
END_VAR
IF NOT bInitialized THEN
	RETURN;
ELSIF NOT fbJson.IsArray(_in_pArrayPointer) THEN
	RETURN;
END_IF

M_AddArrayElement := M_Pushback(_in_pArrayPointer, _in_anyValue);
END_METHOD

(* Adds a new key:value pair to the parameters list and returns a pointer to
	the added value. Supports most primitive types directly.

	If the value is an array, will only add a blank array that must be populated
	manually by calling M_AddArrayElement with the pointer returned by this method. 

	If the value is a struct, will only add a blank struct that must be populated
	manually by calling M_AddStructMember with the pointer returned by this method. 

	Value will be stored as null if the value type is not yet supported. *)
METHOD M_AddParameter : PVOID
VAR_INPUT
	(* Parameter name. *)
	_in_strKey : T_MaxString;
	
	(* Parameter value. *)
	_in_anyValue : ANY;
END_VAR
VAR
	_pJsonMember: Tc3_JsonXml.PVOID;
END_VAR
IF NOT bInitialized THEN
	pJsonDoc := fbJson.NewDocument();
	bInitialized := TRUE;
END_IF

_pJsonMember := THIS^.M_Add(pJsonDoc, _in_strKey, _in_anyValue);

M_AddParameter := _pJsonMember;
END_METHOD

(* Adds a new key:value pair to the parameters list and returns a pointer to
	the added value. Supports most primitive types directly.

	If the value is an array, will only add a blank array that must be populated
	manually by calling M_AddArrayElement with the pointer returned by this method. 

	If the value is a struct, will only add a blank struct that must be populated
	manually by calling M_AddStructMember with the pointer returned by this method. 

	Value will be stored as null if the value type is not yet supported. *)
METHOD M_AddStructMember : PVOID
VAR_INPUT
	(* Pointer to the struct that should be added to. This pointer is returned
		by any M_Add<item> methods that were used to add a struct. *)
	_in_pStructPointer : PVOID;
	
	(* Key to add to the struct. *)
	_in_strKey : T_MaxString;
	
	(* Value to add to the struct. *)
	_in_anyValue : ANY;
END_VAR
IF NOT bInitialized THEN
	M_AddStructMember := 0;
	RETURN;
ELSIF NOT fbJson.IsObject(_in_pStructPointer) THEN
	M_AddStructMember := 0;
	RETURN;
END_IF

M_AddStructMember := M_Add(_in_pStructPointer, _in_strKey, _in_anyValue);
END_METHOD

(* Clears all current parameters. *)
METHOD M_ClearParameters : BOOL
VAR_INPUT
END_VAR
VAR
END_VAR
pJsonDoc := fbJson.NewDocument();
bInitialized := TRUE;
END_METHOD

(* Populates the given parameters list with the added key:value pairs. *)
METHOD M_OutputToParameterList : BOOL
VAR_INPUT
END_VAR
VAR_IN_OUT
	// Parameters list to populate.
	_inout_arrParameters : T_ApiParameterList;
END_VAR
VAR
	_dintParamMin: DINT; // Lower bound of parameters array
	_dintParamMax: DINT; // Upper bound of parameters array
	_dintParamIndex: DINT; // Current parameters array index
	_pJsonIterator: Tc3_JsonXml.PVOID; // Current JSON iterator pointer
	_pJsonIteratorEnd: Tc3_JsonXml.PVOID; // JSON iterator end pointer
	_strName: STRING; // Name of the parameter
	_pValue: Tc3_JsonXml.PVOID; // Pointer to the parameter
	_strValue: T_ApiParamValue; // Parameter value
END_VAR
// Get the array bounds
_dintParamMin := GVL_Api.dintPARAM_LOWER_BOUND;
_dintParamMax := GVL_Api.dintPARAM_UPPER_BOUND;

// Clear the array
FOR _dintParamIndex := _dintParamMin TO _dintParamMax DO
	_inout_arrParameters[_dintParamIndex].strKey := '';
	_inout_arrParameters[_dintParamIndex].strValue := '';
END_FOR

// Initialize the iterators
_dintParamIndex := _dintParamMin;
_pJsonIterator := fbJson.MemberBegin(pJsonDoc);
_pJsonIteratorEnd := fbJson.MemberEnd(pJsonDoc);

// Populate each array member. If there are more parameters than there are
// array members, will stop iterating.
WHILE _pJsonIterator <> _pJsonIteratorEnd AND _dintParamIndex <= _dintParamMax DO
	_strName := fbJson.GetMemberName(_pJsonIterator);
	_pValue := fbJson.GetMemberValue(_pJsonIterator);
	MEMSET(ADR(_strValue),0,SIZEOF(_strValue));
	fbJson.CopyJson(_pValue, _strValue, SIZEOF(_strValue));
	_inout_arrParameters[_dintParamIndex].strKey := _strName;
	_inout_arrParameters[_dintParamIndex].strValue := _strValue;
	_pJsonIterator := fbJson.NextMember(_pJsonIterator);
	_dintParamIndex := _dintParamIndex + 1;
END_WHILE

M_OutputToParameterList := TRUE;
END_METHOD

(* Adds a key:value pair to the given struct. *)
METHOD PRIVATE M_Add : PVOID
VAR_INPUT
	_in_pJsonPointer : PVOID;
	_in_strKey : T_MaxString;
	_in_anyValue : ANY;
END_VAR
VAR
	_pJsonMember: Tc3_JsonXml.PVOID; // Pointer to the added JSON member

	// Supported types
	_pBoolValue:		POINTER TO BOOL;
	_pInt32Value:		POINTER TO DINT;
	_pUint32Value:		POINTER TO UINT;
	_pInt64Value:		POINTER TO LINT;
	_pUint64Value:		POINTER TO ULINT;
	_pDoubleValue:		POINTER TO LREAL;
	_pDateTimeValue:	POINTER TO DATE_AND_TIME;
	_pStringValue:		POINTER TO STRING;
	
	// Converted types
	_pSingleValue:		POINTER TO REAL;
	_pInt16Value:		POINTER TO INT;
	_pInt8Value:		POINTER TO SINT;
	_pUint16Value:		POINTER TO UINT;
	_pUint8Value:		POINTER TO USINT;
	_pByteValue:		POINTER TO BYTE;
	_pWordValue:		POINTER TO WORD;
	_pDwordValue:		POINTER TO DWORD;
	_pLwordValue:		POINTER TO LWORD;
	_pDateValue:		POINTER TO DATE;
	_pTimeValue:		POINTER TO TIME;
	
	// Converted type values
	_lrealSingleValue:	LREAL;
	_dintInt16Value:	DINT;
	_dintInt8Value:		DINT;
	_udintUint16Value:	UDINT;
	_udintUint8Value:	UDINT;
	_udintByteValue:	UDINT;
	_udintWordValue:	UDINT;
	_udintDwordValue:	UDINT;
	_ulintLwordValue:	ULINT;
	_dtDateValue:		DATE_AND_TIME;
	_dtTimeValue:		DATE_AND_TIME;
END_VAR
// Add key-value pair to JSON doc based on type
CASE _in_anyValue.TypeClass OF
	// Supported datatypes
	__SYSTEM.TYPE_CLASS.TYPE_BOOL:
		_pBoolValue := _in_anyValue.pValue;
		_pJsonMember := fbJson.AddBoolMember(_in_pJsonPointer, _in_strKey, _pBoolValue^);
	__SYSTEM.TYPE_CLASS.TYPE_DATEANDTIME:
		_pDateTimeValue := _in_anyValue.pValue;
		_pJsonMember := fbJson.AddDateTimeMember(_in_pJsonPointer, _in_strKey, _pDateTimeValue^);
	__SYSTEM.TYPE_CLASS.TYPE_LREAL:
		_pDoubleValue := _in_anyValue.pValue;
		_pJsonMember := fbJson.AddDoubleMember(_in_pJsonPointer, _in_strKey, _pDoubleValue^);
	__SYSTEM.TYPE_CLASS.TYPE_LINT:
		_pInt64Value := _in_anyValue.pValue;
		_pJsonMember := fbJson.AddInt64Member(_in_pJsonPointer, _in_strKey, _pInt64Value^);
	__SYSTEM.TYPE_CLASS.TYPE_DINT:
		_pInt32Value := _in_anyValue.pValue;
		_pJsonMember := fbJson.AddIntMember(_in_pJsonPointer, _in_strKey, _pInt32Value^);
	__SYSTEM.TYPE_CLASS.TYPE_STRING:
		_pStringValue := _in_anyValue.pValue;
		_pJsonMember := fbJson.AddStringMember(_in_pJsonPointer, _in_strKey, _pStringValue^);
	__SYSTEM.TYPE_CLASS.TYPE_ULINT:
		_pUint64Value := _in_anyValue.pValue;
		_pJsonMember := fbJson.AddUint64Member(_in_pJsonPointer, _in_strKey, _pUint64Value^);
	__SYSTEM.TYPE_CLASS.TYPE_UDINT:
		_pUint32Value := _in_anyValue.pValue;
		_pJsonMember := fbJson.AddUintMember(_in_pJsonPointer, _in_strKey, _pUint32Value^);
		
	// Converted datatypes
	__SYSTEM.TYPE_CLASS.TYPE_REAL:
		_pSingleValue := _in_anyValue.pValue;
		_lrealSingleValue := REAL_TO_LREAL(_pSingleValue^);
		_pJsonMember := fbJson.AddDoubleMember(_in_pJsonPointer, _in_strKey, _lrealSingleValue);
	__SYSTEM.TYPE_CLASS.TYPE_INT:
		_pInt16Value := _in_anyValue.pValue;
		_dintInt16Value := INT_TO_DINT(_pInt16Value^);
		_pJsonMember := fbJson.AddIntMember(_in_pJsonPointer, _in_strKey, _dintInt16Value);
	__SYSTEM.TYPE_CLASS.TYPE_SINT:
		_pInt8Value := _in_anyValue.pValue;
		_dintInt8Value := SINT_TO_DINT(_pInt8Value^);
		_pJsonMember := fbJson.AddIntMember(_in_pJsonPointer, _in_strKey, _dintInt8Value);
	__SYSTEM.TYPE_CLASS.TYPE_UINT:
		_pUint16Value := _in_anyValue.pValue;
		_udintUint16Value := UINT_TO_UDINT(_pUint16Value^);
		_pJsonMember := fbJson.AddUintMember(_in_pJsonPointer, _in_strKey, _udintUint16Value);
	__SYSTEM.TYPE_CLASS.TYPE_USINT:
		_pUint8Value := _in_anyValue.pValue;
		_udintUint8Value := USINT_TO_UDINT(_pUint8Value^);
		_pJsonMember := fbJson.AddUintMember(_in_pJsonPointer, _in_strKey, _udintUint8Value);
	__SYSTEM.TYPE_CLASS.TYPE_BYTE:
		_pByteValue := _in_anyValue.pValue;
		_udintByteValue := BYTE_TO_UDINT(_pByteValue^);
		_pJsonMember := fbJson.AddUintMember(_in_pJsonPointer, _in_strKey, _udintByteValue);
	__SYSTEM.TYPE_CLASS.TYPE_WORD:
		_pWordValue := _in_anyValue.pValue;
		_udintWordValue := WORD_TO_UDINT(_pWordValue^);
		_pJsonMember := fbJson.AddUintMember(_in_pJsonPointer, _in_strKey, _udintWordValue);
	__SYSTEM.TYPE_CLASS.TYPE_DWORD:
		_pDwordValue := _in_anyValue.pValue;
		_udintDwordValue := DWORD_TO_UDINT(_pDwordValue^);
		_pJsonMember := fbJson.AddUintMember(_in_pJsonPointer, _in_strKey, _udintDwordValue);
	__SYSTEM.TYPE_CLASS.TYPE_LWORD:
		_pLwordValue := _in_anyValue.pValue;
		_ulintLwordValue := LWORD_TO_ULINT(_pLwordValue^);
		_pJsonMember := fbJson.AddUint64Member(_in_pJsonPointer, _in_strKey, _ulintLwordValue);
	__SYSTEM.TYPE_CLASS.TYPE_DATE:
		_pDateValue := _in_anyValue.pValue;
		_dtDateValue := DATE_TO_DT(_pDateValue^);
		_pJsonMember := fbJson.AddDateTimeMember(_in_pJsonPointer, _in_strKey, _dtDateValue);
	__SYSTEM.TYPE_CLASS.TYPE_TIME:
		_pTimeValue := _in_anyValue.pValue;
		_dtTimeValue := TIME_TO_DT(_pTimeValue^);
		_pJsonMember := fbJson.AddDateTimeMember(_in_pJsonPointer, _in_strKey, _dtTimeValue);
		
	// Empty objects
	__SYSTEM.TYPE_CLASS.TYPE_ARRAY:
		_pJsonMember := fbJson.AddArrayMember(_in_pJsonPointer, _in_strKey, 0);
	__SYSTEM.TYPE_CLASS.TYPE_USERDEF:
		_pJsonMember := fbJson.AddObjectMember(_in_pJsonPointer, _in_strKey);
		
ELSE
	_pJsonMember := fbJson.AddNullMember(_in_pJsonPointer,_in_strKey);
END_CASE

M_Add := _pJsonMember;
END_METHOD

(* Adds an element to the given array. *)
METHOD PRIVATE M_Pushback : PVOID
VAR_INPUT
	_in_pJsonPointer : PVOID;
	_in_anyValue : ANY;
END_VAR
VAR
	_pJsonMember: Tc3_JsonXml.PVOID;  // Pointer to the added JSON member

	// Supported types
	_pBoolValue:		POINTER TO BOOL;
	_pInt32Value:		POINTER TO DINT;
	_pUint32Value:		POINTER TO UINT;
	_pInt64Value:		POINTER TO LINT;
	_pUint64Value:		POINTER TO ULINT;
	_pDoubleValue:		POINTER TO LREAL;
	_pDateTimeValue:	POINTER TO DATE_AND_TIME;
	_pStringValue:		POINTER TO STRING;
	
	// Converted types
	_pSingleValue:		POINTER TO REAL;
	_pInt16Value:		POINTER TO INT;
	_pInt8Value:		POINTER TO SINT;
	_pUint16Value:		POINTER TO UINT;
	_pUint8Value:		POINTER TO USINT;
	_pByteValue:		POINTER TO BYTE;
	_pWordValue:		POINTER TO WORD;
	_pDwordValue:		POINTER TO DWORD;
	_pLwordValue:		POINTER TO LWORD;
	_pDateValue:		POINTER TO DATE;
	_pTimeValue:		POINTER TO TIME;
	
	// Converted type values
	_lrealSingleValue:	LREAL;
	_dintInt16Value:	DINT;
	_dintInt8Value:		DINT;
	_udintUint16Value:	UDINT;
	_udintUint8Value:	UDINT;
	_udintByteValue:	UDINT;
	_udintWordValue:	UDINT;
	_udintDwordValue:	UDINT;
	_ulintLwordValue:	ULINT;
	_dtDateValue:		DATE_AND_TIME;
	_dtTimeValue:		DATE_AND_TIME;
END_VAR
// Add key-value pair to JSON doc based on type
CASE _in_anyValue.TypeClass OF
	// Supported
	__SYSTEM.TYPE_CLASS.TYPE_BOOL:
		_pBoolValue := _in_anyValue.pValue;
		_pJsonMember := fbJson.PushbackBoolValue(_in_pJsonPointer, _pBoolValue^);
	__SYSTEM.TYPE_CLASS.TYPE_DATEANDTIME:
		_pDateTimeValue := _in_anyValue.pValue;
		_pJsonMember := fbJson.PushbackDateTimeValue(_in_pJsonPointer, _pDateTimeValue^);
	__SYSTEM.TYPE_CLASS.TYPE_LREAL:
		_pDoubleValue := _in_anyValue.pValue;
		_pJsonMember := fbJson.PushbackDoubleValue(_in_pJsonPointer, _pDoubleValue^);
	__SYSTEM.TYPE_CLASS.TYPE_LINT:
		_pInt64Value := _in_anyValue.pValue;
		_pJsonMember := fbJson.PushbackInt64Value(_in_pJsonPointer, _pInt64Value^);
	__SYSTEM.TYPE_CLASS.TYPE_DINT:
		_pInt32Value := _in_anyValue.pValue;
		_pJsonMember := fbJson.PushbackIntValue(_in_pJsonPointer, _pInt32Value^);
	__SYSTEM.TYPE_CLASS.TYPE_STRING:
		_pStringValue := _in_anyValue.pValue;
		_pJsonMember := fbJson.PushbackStringValue(_in_pJsonPointer, _pStringValue^);
	__SYSTEM.TYPE_CLASS.TYPE_ULINT:
		_pUint64Value := _in_anyValue.pValue;
		_pJsonMember := fbJson.PushbackUint64Value(_in_pJsonPointer, _pUint64Value^);
	__SYSTEM.TYPE_CLASS.TYPE_UDINT:
		_pUint32Value := _in_anyValue.pValue;
		_pJsonMember := fbJson.PushbackUintValue(_in_pJsonPointer, _pUint32Value^);
		
	// Converted
	__SYSTEM.TYPE_CLASS.TYPE_REAL:
		_pSingleValue := _in_anyValue.pValue;
		_lrealSingleValue := REAL_TO_LREAL(_pSingleValue^);
		_pJsonMember := fbJson.PushbackDoubleValue(_in_pJsonPointer, _lrealSingleValue);
	__SYSTEM.TYPE_CLASS.TYPE_INT:
		_pInt16Value := _in_anyValue.pValue;
		_dintInt16Value := INT_TO_DINT(_pInt16Value^);
		_pJsonMember := fbJson.PushbackIntValue(_in_pJsonPointer, _dintInt16Value);
	__SYSTEM.TYPE_CLASS.TYPE_SINT:
		_pInt8Value := _in_anyValue.pValue;
		_dintInt8Value := SINT_TO_DINT(_pInt8Value^);
		_pJsonMember := fbJson.PushbackIntValue(_in_pJsonPointer, _dintInt8Value);
	__SYSTEM.TYPE_CLASS.TYPE_UINT:
		_pUint16Value := _in_anyValue.pValue;
		_udintUint16Value := UINT_TO_UDINT(_pUint16Value^);
		_pJsonMember := fbJson.PushbackUintValue(_in_pJsonPointer, _udintUint16Value);
	__SYSTEM.TYPE_CLASS.TYPE_USINT:
		_pUint8Value := _in_anyValue.pValue;
		_udintUint8Value := USINT_TO_UDINT(_pUint8Value^);
		_pJsonMember := fbJson.PushbackUintValue(_in_pJsonPointer, _udintUint8Value);
	__SYSTEM.TYPE_CLASS.TYPE_BYTE:
		_pByteValue := _in_anyValue.pValue;
		_udintByteValue := BYTE_TO_UDINT(_pByteValue^);
		_pJsonMember := fbJson.PushbackUintValue(_in_pJsonPointer, _udintByteValue);
	__SYSTEM.TYPE_CLASS.TYPE_WORD:
		_pWordValue := _in_anyValue.pValue;
		_udintWordValue := WORD_TO_UDINT(_pWordValue^);
		_pJsonMember := fbJson.PushbackUintValue(_in_pJsonPointer, _udintWordValue);
	__SYSTEM.TYPE_CLASS.TYPE_DWORD:
		_pDwordValue := _in_anyValue.pValue;
		_udintDwordValue := DWORD_TO_UDINT(_pDwordValue^);
		_pJsonMember := fbJson.PushbackUintValue(_in_pJsonPointer, _udintDwordValue);
	__SYSTEM.TYPE_CLASS.TYPE_LWORD:
		_pLwordValue := _in_anyValue.pValue;
		_ulintLwordValue := LWORD_TO_ULINT(_pLwordValue^);
		_pJsonMember := fbJson.PushbackUint64Value(_in_pJsonPointer, _ulintLwordValue);
	__SYSTEM.TYPE_CLASS.TYPE_DATE:
		_pDateValue := _in_anyValue.pValue;
		_dtDateValue := DATE_TO_DT(_pDateValue^);
		_pJsonMember := fbJson.PushbackDateTimeValue(_in_pJsonPointer, _dtDateValue);
	__SYSTEM.TYPE_CLASS.TYPE_TIME:
		_pTimeValue := _in_anyValue.pValue;
		_dtTimeValue := TIME_TO_DT(_pTimeValue^);
		_pJsonMember := fbJson.PushbackDateTimeValue(_in_pJsonPointer, _dtTimeValue);
	
	// Objects
	__SYSTEM.TYPE_CLASS.TYPE_ARRAY:
		_pJsonMember := fbJson.PushbackJsonValue(_in_pJsonPointer, '[]');
	__SYSTEM.TYPE_CLASS.TYPE_USERDEF:
		_pJsonMember := fbJson.PushbackJsonValue(_in_pJsonPointer, '{}');
ELSE
	_pJsonMember := fbJson.PushbackNullValue(_in_pJsonPointer);
END_CASE

M_Pushback := _pJsonMember;
END_METHOD

METHOD M_ParseBool : BOOL
VAR_INPUT
	(* Pointer to the value. *)
	_in_pValuePointer : PVOID;
END_VAR
IF _in_pValuePointer = 0 THEN
	THIS^.M_LogWarning('Invalid pointer in M_ParseBool!');
	RETURN;
END_IF
IF fbJson.IsBool(_in_pValuePointer) THEN
	M_ParseBool := fbJson.GetBool(_in_pValuePointer);
END_IF
END_METHOD

METHOD M_ParseDateTime : DATE_AND_TIME
VAR_INPUT
	(* Pointer to the value. *)
	_in_pValuePointer : PVOID;
END_VAR
IF _in_pValuePointer = 0 THEN
	THIS^.M_LogWarning('Invalid pointer in M_ParseDateTime!');
	RETURN;
END_IF
IF fbJson.IsISO8601TimeFormat(_in_pValuePointer) THEN
	M_ParseDateTime := fbJson.GetDateTime(_in_pValuePointer);
END_IF
END_METHOD

METHOD M_ParseDouble : LREAL
VAR_INPUT
	(* Pointer to the value. *)
	_in_pValuePointer : PVOID;
END_VAR
IF _in_pValuePointer = 0 THEN
	THIS^.M_LogWarning('Invalid pointer in M_ParseDouble!');
	RETURN;
END_IF
IF fbJson.IsDouble(_in_pValuePointer) THEN
	M_ParseDouble := fbJson.GetDouble(_in_pValuePointer);
END_IF
END_METHOD

METHOD M_ParseInt : DINT
VAR_INPUT
	(* Pointer to the value. *)
	_in_pValuePointer : PVOID;
END_VAR
IF _in_pValuePointer = 0 THEN
	THIS^.M_LogWarning('Invalid pointer in M_ParseInt!');
	RETURN;
END_IF
IF fbJson.IsInt(_in_pValuePointer) THEN
	M_ParseInt := fbJson.GetInt(_in_pValuePointer);
END_IF
END_METHOD

METHOD M_ParseInt64 : LINT
VAR_INPUT
	(* Pointer to the value. *)
	_in_pValuePointer : PVOID;
END_VAR
IF _in_pValuePointer = 0 THEN
	THIS^.M_LogWarning('Invalid pointer in M_ParseInt64!');
	RETURN;
END_IF
IF fbJson.IsInt64(_in_pValuePointer) THEN
	M_ParseInt64 := fbJson.GetInt64(_in_pValuePointer);
END_IF
END_METHOD

METHOD M_ParseString : T_MaxString
VAR_INPUT
	(* Pointer to the value. *)
	_in_pValuePointer : PVOID;
END_VAR
IF _in_pValuePointer = 0 THEN
	THIS^.M_LogWarning('Invalid pointer in M_ParseString!');
	RETURN;
END_IF
IF fbJson.IsString(_in_pValuePointer) THEN
	M_ParseString := fbJson.GetString(_in_pValuePointer);
END_IF
END_METHOD

METHOD M_ParseUint : UDINT
VAR_INPUT
	(* Pointer to the value. *)
	_in_pValuePointer : PVOID;
END_VAR
IF _in_pValuePointer = 0 THEN
	THIS^.M_LogWarning('Invalid pointer in M_ParseUint!');
	RETURN;
END_IF
IF fbJson.IsUint(_in_pValuePointer) THEN
	M_ParseUInt := fbJson.GetUint(_in_pValuePointer);
END_IF
END_METHOD

METHOD M_ParseUint64 : ULINT
VAR_INPUT
	(* Pointer to the value. *)
	_in_pValuePointer : PVOID;
END_VAR
IF _in_pValuePointer = 0 THEN
	THIS^.M_LogWarning('Invalid pointer in M_ParseUint64!');
	RETURN;
END_IF
IF fbJson.IsUint64(_in_pValuePointer) THEN
	M_ParseUInt64 := fbJson.GetUint64(_in_pValuePointer);
END_IF
END_METHOD

(* Returns a pointer to the value of the given array index inside of the
	array given by the pointer. Use the relevant M_Parse<type> method
	to get the data from the value. *)
METHOD M_GetArrayElement : PVOID
VAR_INPUT
	(* Pointer to the struct to get the member from. *)
	_in_pArrayPointer : PVOID;
	(* Index of the element to get. *)
	_in_udintIndex : UDINT;
END_VAR
IF bInitialized THEN
	M_GetArrayElement := fbJson.GetArrayValueByIdx(_in_pArrayPointer, _in_udintIndex);
END_IF
END_METHOD

(* Returns a pointer to the value of the requested parameter. Use the relevant
	M_Parse<type> method to get the data from the value, or M_GetStructMember
	or M_GetArrayElement if the value is a struct or array respectively. *)
METHOD M_GetParameter : PVOID
VAR_INPUT
	(* Name of the parameter to get. *)
	_in_strName : T_MaxString;
END_VAR
M_GetParameter := M_GetStructMember(pJsonDoc, _in_strName);
END_METHOD

(* Returns a pointer to the value of the given parameter inside of the
	struct given by the pointer. Use the relevant M_Parse<type> method
	to get the data from the value. *)
METHOD M_GetStructMember : PVOID
VAR_INPUT
	(* Pointer to the struct to get the member from. *)
	_in_pStructPointer : PVOID;
	(* Name of the parameter to get. *)
	_in_strName : T_MaxString;
END_VAR
IF bInitialized THEN
	M_GetStructMember := fbJson.FindMember(_in_pStructPointer, _in_strName);
END_IF
END_METHOD

METHOD M_LoadFromParameterList : BOOL
VAR_INPUT
END_VAR
VAR_IN_OUT
	// Parameters list to load into the function block.
	_inout_arrParameters : T_ApiParameterList;
END_VAR
VAR
	_dintParamMin: DINT; // Lower bound of the parameters array
	_dintParamMax: DINT; // Upper bound of the parameters array
	_dintParamIndex: DINT; // Current index of the parameters array
	_strKey: STRING(255); // Name of the parameter
	_strValue: T_ApiParamValue; // Value of the parameter
END_VAR
// Clear the JSON doc
pJsonDoc := fbJson.NewDocument();
bInitialized := TRUE;

// Get the array bounds
_dintParamMin := GVL_Api.dintPARAM_LOWER_BOUND;
_dintParamMax := GVL_Api.dintPARAM_UPPER_BOUND;

// Populate the JSON document
FOR _dintParamIndex := _dintParamMin TO _dintParamMax DO
	_strKey := _inout_arrParameters[_dintParamIndex].strKey;
	_strValue := _inout_arrParameters[_dintParamIndex].strValue;
	IF LEN(_strKey) > 0 THEN
		fbJson.AddJsonMember(pJsonDoc, _strKey, _strValue);
	END_IF
END_FOR

M_LoadFromParameterList := TRUE;
END_METHOD

END_FUNCTION_BLOCK

// Interfaces/Obsolete/I_ModularAPI
INTERFACE I_ModularAPI

(* Calls a method on the modular API, and returns true once
	the result of the method is received. *)
METHOD M_CallMethod : BOOL
VAR_INPUT
	(* ID of the module the method is being routed to. *)
	strModuleId: T_MaxString;
	
	(* Name of the API method that will be called. *)
	strMethodName: T_MaxString;
	
	(* An array of array of strings representing the name:value pair
		for all of the required method parameters. *)
	arrParameters: T_ApiMethodParameters;
END_VAR
VAR_OUTPUT
	(* Should be TRUE if the method executed without error. *)
	bSuccessful: BOOL;
	
	(* The return value of the method. *)
	strReturnValue: T_MaxString;
	
	(* Name:value pairs for any outputs of the method. *)
	arrOutputValues: T_ApiMethodParameters;
END_VAR
END_METHOD

(* Should return TRUE if there is a method in this interface that
	is executing. *)
PROPERTY P_bApiBusy : BOOL
GET
END_GET
END_PROPERTY

END_INTERFACE

// Project Information/F_GetCompany
// This function has been automatically generated from the project information.
{attribute 'signature_flag' := '1073741824'}
{attribute 'TcGenerated'}
{attribute 'no-analysis'}
FUNCTION F_GetCompany : WSTRING
VAR_INPUT
	
END_VAR

F_GetCompany := "Sensata Technologies";

END_FUNCTION

// Project Information/F_GetTitle
// This function has been automatically generated from the project information.
{attribute 'signature_flag' := '1073741824'}
{attribute 'TcGenerated'}
{attribute 'no-analysis'}
FUNCTION F_GetTitle : WSTRING
VAR_INPUT
	
END_VAR

F_GetTitle := "Sensata_Utilities";

END_FUNCTION

// Project Information/F_GetVersion
// This function has been automatically generated from the project information.
{attribute 'signature_flag' := '1073741824'}
{attribute 'TcGenerated'}
{attribute 'no-analysis'}
FUNCTION F_GetVersion : ST_LibVersion
VAR_INPUT
	
END_VAR

F_GetVersion.iMajor := 0;
F_GetVersion.iMinor := 0;
F_GetVersion.iBuild := 1;
F_GetVersion.iRevision := 0;

END_FUNCTION
